(* CODESYS project GVL_MULTI_TYPE.gvl.xml

Project tree, tasks and I/O mapping:
  global variables GVL_MULTI_TYPE
*)

// GVL_MULTI_TYPE
{attribute 'qualified_only'}
VAR_GLOBAL
	Config       : ST_MULTI_TYPE_CONFIG; // Активная конфигурация типов продукции
	ConfigStatus : ST_MULTI_TYPE_CONFIG_STATUS; // Разрешения редактирования конфигурации
	CycleStatus  : ST_CELL_CYCLE_STATUS; // Диагностика универсального автомата ячейки
END_VAR
